(* PLC project SafeLOGIC, BrAutomation SafeDESIGNER  5.24.1.0 *)
(* stored: companyURL http://www.br-automation.com, creationDateTime Mon Aug 11 10:46:45 2025 *)

PROGRAM DEVIATION
  VAR  (* added by the conversion: wires and edge detectors of the diagram *)
    _AND_S34_OUT : ANY;
  END_VAR

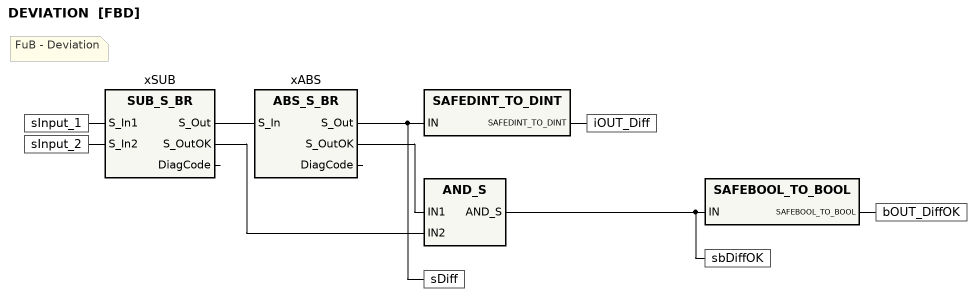
(* FBD diagram, written out as Structured Text *)
(* FuB - Deviation *)
xSUB(S_In1 := sInput_1, S_In2 := sInput_2);
xABS(S_In := xSUB.S_Out);
iOUT_Diff := SAFEDINT_TO_DINT(xABS.S_Out);
_AND_S34_OUT := AND_S(xABS.S_OutOK, xSUB.S_OutOK);
sbDiffOK := _AND_S34_OUT;
sDiff := xABS.S_Out;
bOUT_DiffOK := SAFEBOOL_TO_BOOL(_AND_S34_OUT);
END_PROGRAM
